{attribute 'no_explicit_call' := 'do not call this function block directly'} 
FUNCTION_BLOCK WaitVariableValueActivity EXTENDS Activity IMPLEMENTS IWaitVariableValueActivity
VAR
	{attribute 'OPC.UA.DA' := '0'}
	_ClassName : STRING := __POUNAME();
	
	{attribute 'OPC.UA.DA' := '0'}
	_Condition : VariableHasValueCondition;
END_VAR

{attribute 'monitoring' := 'call'}
PROPERTY ClassName : STRING
GET
ClassName := _ClassName;
END_GET
END_PROPERTY

METHOD Configure
VAR_INPUT
	monitoredVariableName : STRING;
	referenceValue : ANY; 
END_VAR
VAR
	variableNameEmptyException : Core.ArgumentOutOfRangeException;
	referenceValueNullException : Core.ArgumentNullException; 
END_VAR
IF monitoredVariableName = '' THEN
	variableNameEmptyException.Throw(CurrentNamespace.Name, ClassName, __POUNAME(), __POSITION(), 'monitoredVariableName', monitoredVariableName);
END_IF

IF referenceValue.pValue = 0 OR_ELSE referenceValue.diSize = 0 THEN
	referenceValueNullException.Throw(CurrentNamespace.Name, ClassName, __POUNAME(), __POSITION(), 'referenceValue');
END_IF

_Condition.InternalConfigure(monitoredVariableName, referenceValue);
END_METHOD

{attribute 'monitoring' := 'call'}
PROPERTY MonitoredVariableName : STRING
GET
MonitoredVariableName := _Condition.MonitoredVariableName;
END_GET
END_PROPERTY

{attribute 'monitoring' := 'call'}
PROPERTY Name : WSTRING
GET
Name := SEL(_Name = "", _Name, TO_WSTRING(ClassName));
END_GET
SET
_Name := Name;
END_SET
END_PROPERTY

METHOD PROTECTED OnAborting 
VAR_INPUT
	start : BOOL;
END_VAR
VAR_OUTPUT
	done : BOOL;
END_VAR
done := TRUE;
END_METHOD

METHOD PROTECTED OnRunning 
VAR_INPUT
	start : BOOL;
END_VAR
VAR_OUTPUT
	done : BOOL;
END_VAR
VAR
	workflowVariable : Core.GENERIC_VALUE;
END_VAR
done := _Condition.Evaluate(Workflow, THIS^);
END_METHOD

{attribute 'monitoring' := 'call'}
PROPERTY ReferenceValue : __SYSTEM.AnyType
GET
ReferenceValue := _Condition.ReferenceValue;
END_GET
END_PROPERTY

{attribute 'monitoring' := 'call'}
PROPERTY FINAL Size : ULINT
GET
Size := XSIZEOF(THIS^);
END_GET
END_PROPERTY

END_FUNCTION_BLOCK

(* stored: Version 1.1.0.1
   POU WaitVariableValueActivity: Id {42ec5adb-5b33-4f97-b06e-abb67d1deb50}, SpecialFunc None
   Folder Overriden: Id {e869c370-97ea-4440-962a-299b7c76714e}
   Property ClassName: Id {9255cdcc-cc75-4b54-a049-e35c44af441b}
   Get Get: Id {75ca8576-7cf6-486a-8444-bb56a0b67c7f}
   Method Configure: Id {e9d27d0c-0ec6-4b8c-b0ee-313d596c221a}
   Property MonitoredVariableName: Id {9c3073b8-fb93-4527-9e2b-1b57a617b10a}
   Get Get: Id {53a3a5d7-b81b-4c1b-b3d8-075259b5275f}
   Property Name: Id {4d113431-1828-49a5-adc6-543ca94a7ab4}
   Get Get: Id {8d709444-a2cc-4b65-bd92-b4309202c126}
   Set Set: Id {a3efb13e-325e-4300-a464-c1f28cdc1d7f}
   Method OnAborting: Id {5b13f21b-b6c4-416d-8afb-2c568361ecfa}
   Method OnRunning: Id {fb76f864-38cb-421c-8f70-82cee258b114}
   Property ReferenceValue: Id {10cce365-b3cc-47cf-93c2-3f365e8252c3}
   Get Get: Id {5491a43e-b72e-479a-af20-3f1aed552bf3}
   Property Size: Id {b5de74a5-a12f-46ac-a733-2c588aa0097f}
   Get Get: Id {080d625a-a924-4e07-839e-cbdd7c0560e8} *)
